FUNCTION calculateTargetTemperatureOn : REAL
VAR_INPUT
	photovoltaicSurplus			: BOOL;
END_VAR

IF (photovoltaicSurplus) THEN
    calculateTargetTemperatureOn := GVL.configValues.targetTemperatureOnPV;
ELSE
    calculateTargetTemperatureOn := GVL.configValues.targetTemperatureOn;
END_IF;

END_FUNCTION

(* stored: Version 1.1.0.1
   POU calculateTargetTemperatureOn: Id {3996f331-fc86-48cb-a3ea-01427f983d4a}, SpecialFunc None *)
